% RSLogix 500 project TRAFFIC CONTROL_BAK005.RSS, saved by version 8.30.00.16 %
PROJECT "UNTITLED"    % processor: Bul.1763 MicroLogix 1100 Series B %

PROGRAM FILES
  LAD 2   11 rungs

DATA FILES
  O0 OUTPUT  4 elements
  I1 INPUT  6 elements
  S2 STATUS  66 elements
  B3 BINARY  1 elements
  T4 TIMER  4 elements
  C5 COUNTER  1 elements
  R6 CONTROL  1 elements
  N7 INTEGER  1 elements
  F8 FLOAT  1 elements

LADDER 2
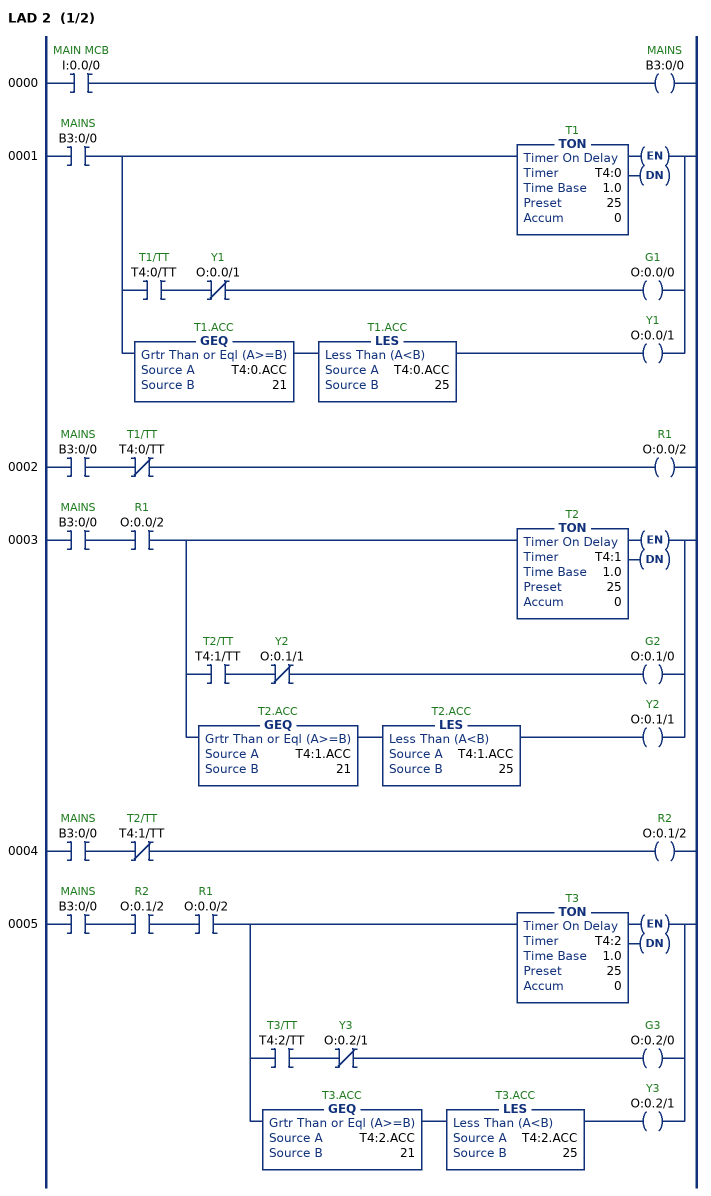
% Rung: 0 %
SOR XIC I:0.0/0 OTE B3:0/0 EOR
%   I:0.0/0  "MAIN MCB" %
%   B3:0/0  "MAINS" %
% Rung: 1 %
SOR XIC B3:0/0 BST TON T4:0 1.0 25 0 NXB BST XIC T4:0/TT XIO O:0.0/1 OTE O:0.0/0 NXB GEQ T4:0.ACC 21 LES T4:0.ACC 25 OTE O:0.0/1 BND BND EOR
%   B3:0/0  "MAINS" %
%   T4:0  T1 %
%   O:0.0/1  "Y1" %
%   O:0.0/0  "G1" %
% Rung: 2 %
SOR XIC B3:0/0 XIO T4:0/TT OTE O:0.0/2 EOR
%   B3:0/0  "MAINS" %
%   T4:0  T1 %
%   O:0.0/2  "R1" %
% Rung: 3 %
SOR XIC B3:0/0 XIC O:0.0/2 BST TON T4:1 1.0 25 0 NXB BST XIC T4:1/TT XIO O:0.1/1 OTE O:0.1/0 NXB GEQ T4:1.ACC 21 LES T4:1.ACC 25 OTE O:0.1/1 BND BND EOR
%   B3:0/0  "MAINS" %
%   O:0.0/2  "R1" %
%   T4:1  T2 %
%   O:0.1/1  "Y2" %
%   O:0.1/0  "G2" %
% Rung: 4 %
SOR XIC B3:0/0 XIO T4:1/TT OTE O:0.1/2 EOR
%   B3:0/0  "MAINS" %
%   T4:1  T2 %
%   O:0.1/2  "R2" %
% Rung: 5 %
SOR XIC B3:0/0 XIC O:0.1/2 XIC O:0.0/2 BST TON T4:2 1.0 25 0 NXB BST XIC T4:2/TT XIO O:0.2/1 OTE O:0.2/0 NXB GEQ T4:2.ACC 21 LES T4:2.ACC 25 OTE O:0.2/1 BND BND EOR
%   B3:0/0  "MAINS" %
%   O:0.1/2  "R2" %
%   O:0.0/2  "R1" %
%   T4:2  T3 %
%   O:0.2/1  "Y3" %
%   O:0.2/0  "G3" %

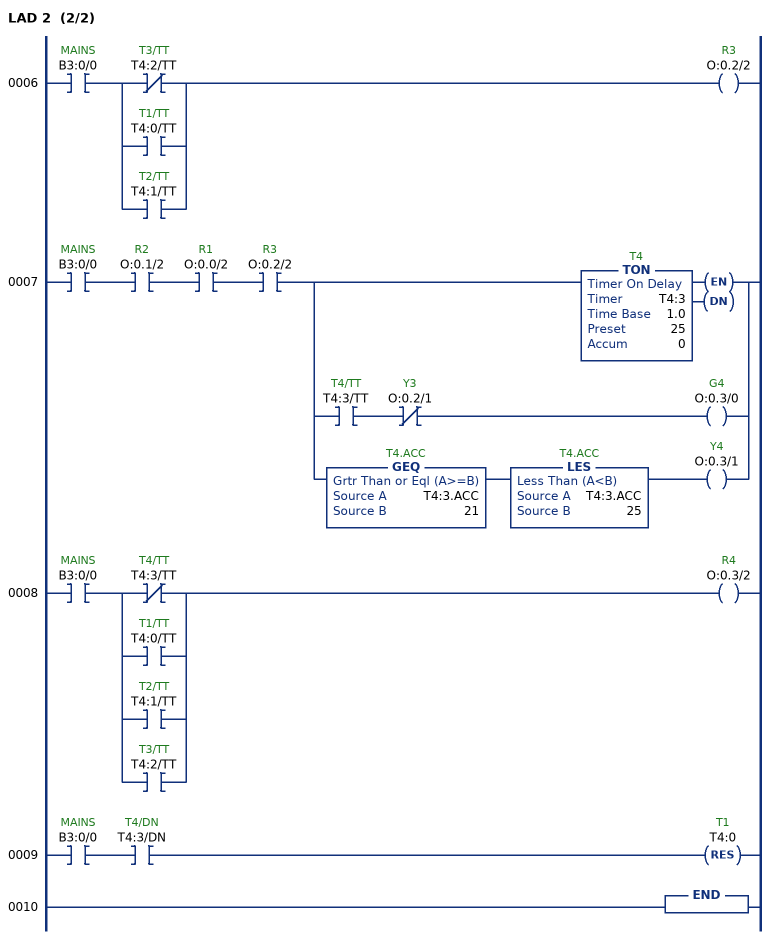
% Rung: 6 %
SOR XIC B3:0/0 BST XIO T4:2/TT NXB BST XIC T4:0/TT NXB XIC T4:1/TT BND BND OTE O:0.2/2 EOR
%   B3:0/0  "MAINS" %
%   T4:2  T3 %
%   T4:0  T1 %
%   T4:1  T2 %
%   O:0.2/2  "R3" %
% Rung: 7 %
SOR XIC B3:0/0 XIC O:0.1/2 XIC O:0.0/2 XIC O:0.2/2 BST TON T4:3 1.0 25 0 NXB BST XIC T4:3/TT XIO O:0.2/1 OTE O:0.3/0 NXB GEQ T4:3.ACC 21 LES T4:3.ACC 25 OTE O:0.3/1 BND BND EOR
%   B3:0/0  "MAINS" %
%   O:0.1/2  "R2" %
%   O:0.0/2  "R1" %
%   O:0.2/2  "R3" %
%   T4:3  T4 %
%   O:0.2/1  "Y3" %
%   O:0.3/0  "G4" %
%   O:0.3/1  "Y4" %
% Rung: 8 %
SOR XIC B3:0/0 BST XIO T4:3/TT NXB BST XIC T4:0/TT NXB BST XIC T4:1/TT NXB XIC T4:2/TT BND BND BND OTE O:0.3/2 EOR
%   B3:0/0  "MAINS" %
%   T4:3  T4 %
%   T4:0  T1 %
%   T4:1  T2 %
%   T4:2  T3 %
%   O:0.3/2  "R4" %
% Rung: 9 %
SOR XIC B3:0/0 XIC T4:3/DN RES T4:0 EOR
%   B3:0/0  "MAINS" %
%   T4:3  T4 %
%   T4:0  T1 %
% Rung: 10 %
SOR END EOR

DATA TABLE (non-zero values as saved)
DATA T4
% .PRE .ACC %
% T4:0 % 25 0
% T4:1 % 25 0
% T4:2 % 25 0
% T4:3 % 25 0
